   VAR
      s_FB_ItemError { ExternalAccessible := 'False'; ExternalVisible := 'False'; ExternalWritable := 'False'; S7_SetPoint := 'False'} : "FB_ItemError";   // Item error block's instance
      s_FB_ItemStatus { ExternalAccessible := 'False'; ExternalVisible := 'False'; ExternalWritable := 'False'; S7_SetPoint := 'False'} : "FB_ItemStatus";   // Item status block's instance
      ss_FIFOStatus { ExternalAccessible := 'False'; ExternalVisible := 'False'; ExternalWritable := 'False'; S7_SetPoint := 'False'} : "UDT_FifoStatus";   // Status structure
      s_UDT_Message { ExternalAccessible := 'False'; ExternalVisible := 'False'; ExternalWritable := 'False'; S7_SetPoint := 'False'} : "UDT_MessageV2";   // Message
      s_UDT_CodingBeltModesStatusOld { ExternalAccessible := 'False'; ExternalVisible := 'False'; ExternalWritable := 'False'; S7_SetPoint := 'False'} : "UDT_CodingBeltModesStatus";   // CodingBeltModes status structure
      s_UDT_ItemError { ExternalAccessible := 'False'; ExternalVisible := 'False'; ExternalWritable := 'False'; S7_SetPoint := 'False'} : "UDT_ItemError";   // Item error message body structure
      s_UDT_ItemStatus { ExternalAccessible := 'False'; ExternalVisible := 'False'; ExternalWritable := 'False'; S7_SetPoint := 'False'} : "UDT_ItemStatus";   // Item status message body structure
      s_R_TRIG_Connection {InstructionName := 'R_TRIG'; LibVersion := '1.0'; ExternalAccessible := 'False'; ExternalVisible := 'False'; ExternalWritable := 'False'; S7_SetPoint := 'False'} : R_TRIG;   // Rising edge trigger connection reastablished
      s_F_TRIG_SendAllErrors {InstructionName := 'F_TRIG'; LibVersion := '1.0'; ExternalAccessible := 'False'; ExternalVisible := 'False'; ExternalWritable := 'False'; S7_SetPoint := 'False'} : F_TRIG;   // Falling edge trigger from signal send all errors
      sdi_Code { ExternalAccessible := 'False'; ExternalVisible := 'False'; ExternalWritable := 'False'} : DInt;   // Error code
      si_ItemStatus { ExternalAccessible := 'False'; ExternalVisible := 'False'; ExternalWritable := 'False'} : Int;   // Item status
      ii_ErrorNumber { ExternalAccessible := 'False'; ExternalVisible := 'False'; ExternalWritable := 'False'} : Int;   // Counter Error Number
      si_State { ExternalAccessible := 'False'; ExternalVisible := 'False'; ExternalWritable := 'False'} : Int;   // Error state
      sx_ItemErrorMessageReq { ExternalAccessible := 'False'; ExternalVisible := 'False'; ExternalWritable := 'False'} : Bool;   // Item error message required
      sx_ItemStatusMessageReq { ExternalAccessible := 'False'; ExternalVisible := 'False'; ExternalWritable := 'False'} : Bool;   // Item status message required
      sx_SendAllProcedure { ExternalAccessible := 'False'; ExternalVisible := 'False'; ExternalWritable := 'False'} : Bool;   // Send all procedure
      sx_FIFOError { ExternalAccessible := 'False'; ExternalVisible := 'False'; ExternalWritable := 'False'} : Bool;   // FIFO error
      sx_FIFOWarning { ExternalAccessible := 'False'; ExternalVisible := 'False'; ExternalWritable := 'False'} : Bool;   // FIFO warning
      sx_ItemErrorBlockError { ExternalAccessible := 'False'; ExternalVisible := 'False'; ExternalWritable := 'False'} : Bool;   // Item error block error
      sx_ItemErrorBlockWarning { ExternalAccessible := 'False'; ExternalVisible := 'False'; ExternalWritable := 'False'} : Bool;   // Item error block warning
      sx_ItemStatusBlockError { ExternalAccessible := 'False'; ExternalVisible := 'False'; ExternalWritable := 'False'} : Bool;   // Item status block error
      sx_ItemStatusBlockWarning { ExternalAccessible := 'False'; ExternalVisible := 'False'; ExternalWritable := 'False'} : Bool;   // Item status block warning
   END_VAR


BEGIN
	(*
	----------------------------------------------------------------------------------------
	|                                                                                      |
	|  Copyright  2023             FORTNA Europe BV                                        |
	|  All Rights Reserved         Netherlands                                             |
	|                                                                                      |
	----------------------------------------------------------------------------------------
	Version history:
	Date        | Version   | Author       | Remark
	----------------------------------------------------------------------------------------
	26/04/2023  | 1.0       | M. Diebel   | Release TIA 17  | DHL Munich 2023
	06/10/2023  | 1.1       | M. Diebel   | Status handling | DHL Munich 2023
	13/03/2023  | 1.2       | S. Nieswiec  | Updated for new Baseline
	*)


	REGION 1 - Initialize message required signals

	    #sx_ItemErrorMessageReq := FALSE;
	    #sx_ItemStatusMessageReq := FALSE;

	    // On connection reestablish send last remembered status and error state ( status only when it's diffrent then 0 )
	    #s_R_TRIG_Connection(CLK := #ix_MFCConnected);

	    IF #s_R_TRIG_Connection.Q AND #si_ItemStatus <> 0
	    THEN
	        #sx_ItemStatusMessageReq := TRUE;
	    END_IF;

	    IF #s_R_TRIG_Connection.Q
	    THEN
	        #sx_ItemErrorMessageReq := TRUE;
	    END_IF;

	    // Prepare trigger on the collective reset signal.
	    #s_F_TRIG_SendAllErrors(CLK := #ix_SendAllErrorsState);

	    // When collective reset will go down, start send every equipment errors.
	    IF #s_F_TRIG_SendAllErrors.Q AND NOT #sx_SendAllProcedure
	    THEN
	        #ii_ErrorNumber := 0;
	        #sx_SendAllProcedure := TRUE;
	    END_IF;

	END_REGION

	REGION 2 - FIFO header status update

	    // Mode 'S' - FIFO register status update.
	    "FC_Fifo"(ic_Mode := 'S',
	              qUDT_Status => #ss_FIFOStatus,
	              qx_Error => #sx_FIFOError,
	              qx_Warning => #sx_FIFOWarning,
	              iqv_Data := #s_UDT_Message,
	              iqUDT_FifoHeader := #iq_UDT_FifoHeader,
	              iqv_DataBuffer := #iqs_FifoData);

	END_REGION

	REGION 3 - Prepare message data

	    // When there is no reset errors command, update errors.
	    IF NOT #ix_CollectiveReset
	        AND NOT #ss_FIFOStatus.FifoPreFull
	    THEN

	        // Status
	        IF (#i_UDT_CodingBeltModesStatus.Status <> #s_UDT_CodingBeltModesStatusOld.Status OR (#sx_SendAllProcedure AND #ii_ErrorNumber = 0))
	        THEN
	            #sx_ItemStatusMessageReq := TRUE;
	            #si_ItemStatus := #i_UDT_CodingBeltModesStatus.Status;
	            #s_UDT_CodingBeltModesStatusOld.Status := #i_UDT_CodingBeltModesStatus.Status;
	            #sx_SendAllProcedure := FALSE;
	        END_IF;


	        IF (#i_UDT_CodingBeltModesStatus.Specific.GeneralError <> #s_UDT_CodingBeltModesStatusOld.Specific.GeneralError AND NOT #sx_SendAllProcedure)
	            OR (#sx_SendAllProcedure AND #ii_ErrorNumber = 0)
	        THEN
	            #sdi_Code := "DB_MFC_ErrorCode".CodingBeltModes.GeneralError;
	            #si_State := BOOL_TO_INT(#i_UDT_CodingBeltModesStatus.Specific.GeneralError);
	            #s_UDT_CodingBeltModesStatusOld.Specific.GeneralError := #i_UDT_CodingBeltModesStatus.Specific.GeneralError;
	            #sx_ItemErrorMessageReq := TRUE;
	            #ii_ErrorNumber += 1;
	        ELSIF (#i_UDT_CodingBeltModesStatus.Specific.ConfigurationError <> #s_UDT_CodingBeltModesStatusOld.Specific.ConfigurationError AND NOT #sx_SendAllProcedure)
	            OR (#sx_SendAllProcedure AND #ii_ErrorNumber = 1)
	        THEN
	            #sdi_Code := "DB_MFC_ErrorCode".CodingBeltModes.ConfigurationError;
	            #si_State := BOOL_TO_INT(#i_UDT_CodingBeltModesStatus.Specific.ConfigurationError);
	            #s_UDT_CodingBeltModesStatusOld.Specific.ConfigurationError := #i_UDT_CodingBeltModesStatus.Specific.ConfigurationError;
	            #sx_ItemErrorMessageReq := TRUE;
	            #ii_ErrorNumber += 1;
	            #sx_SendAllProcedure := FALSE;
	        END_IF;

	    END_IF;

	END_REGION

	REGION 4 - Write message components to the item error structure

	    #s_UDT_ItemError.ItemNumber := #i_UDT_EquipmentNumber;
	    #s_UDT_ItemError.Error := #sdi_Code;
	    #s_UDT_ItemError.State := #si_State;
	    #s_UDT_ItemError.Masked := 1;

	END_REGION

	REGION 5 - Write message components to the item status structure

	    #s_UDT_ItemStatus.Group := #i_UDT_EquipmentNumber.Group;
	    #s_UDT_ItemStatus.Node := #i_UDT_EquipmentNumber.Node;
	    #s_UDT_ItemStatus.Status := #si_ItemStatus;

	END_REGION

	REGION 6 - Prepare messages to the MFC

	    // If item error message required signal is set, prepare the item error message.
	    IF (#sx_ItemErrorMessageReq)
	    THEN
	        #s_FB_ItemError(i_UDT_ItemErrorBody := #s_UDT_ItemError,
	                        ii_MessageGroup := 1,
	                        ix_FlagRetry := FALSE,
	                        idi_TimeSpan := 0,
	                        qx_Error => #sx_ItemErrorBlockError,
	                        qx_Warning => #sx_ItemErrorBlockWarning,
	                        iq_UDT_FifoHeader := #iq_UDT_FifoHeader,
	                        iqs_FifoData := #iqs_FifoData,
	                        iqdi_MessageSequenceNumber := #iqdi_MessageSequenceNumber);
	    END_IF;

	    // If item status message required signal is set, prepare the item error message.
	    IF (#sx_ItemStatusMessageReq)
	    THEN
	        #s_FB_ItemStatus(i_UDT_ItemStatusBody := #s_UDT_ItemStatus,
	                         ii_MessageGroup := 1,
	                         ix_FlagRetry := FALSE,
	                         idi_TimeSpan := 0,
	                         qx_Error => #sx_ItemStatusBlockError,
	                         qx_Warning => #sx_ItemStatusBlockWarning,
	                         iq_UDT_FifoHeader := #iq_UDT_FifoHeader,
	                         iqs_FifoData := #iqs_FifoData,
	                         iqdi_MessageSequenceNumber := #iqdi_MessageSequenceNumber);
	    END_IF;

	END_REGION

	REGION 7 - Write outputs

	    // Prepare collective output error.
	    #qx_Error :=
	    #sx_ItemErrorBlockError
	    OR #sx_ItemStatusBlockError
	    OR #sx_FIFOError;

	    // Prepare collective output warning.
	    #qx_Warning :=
	    #sx_ItemErrorBlockWarning
	    OR #sx_ItemStatusBlockWarning
	    OR #sx_FIFOWarning;

	END_REGION




END_FUNCTION_BLOCK

FUNCTION_BLOCK "FB_MFC_Visu_PECUpdate_Status"
{ S7_Optimized_Access := 'TRUE' }
VERSION : 2.0
// ATTRIBUTES
// AUTO_NUMBER = True
// BLOCK_NUMBER = 249
// END_ATTRIBUTES
   VAR_INPUT
      ix_SendAllErrorsState { ExternalAccessible := 'False'; ExternalVisible := 'False'; ExternalWritable := 'False'} : Bool;   // True - update all the messages
      ix_MFCConnected { ExternalAccessible := 'False'; ExternalVisible := 'False'; ExternalWritable := 'False'} : Bool;   // True - A connection to the MFC has been established
      ix_CollectiveReset { ExternalAccessible := 'False'; ExternalVisible := 'False'; ExternalWritable := 'False'} : Bool;   // True - Collective reset command of all system controls
      i_UDT_PECUpdateStatus { ExternalAccessible := 'False'; ExternalVisible := 'False'; ExternalWritable := 'False'} : "UDT_PECUpdateStatus";   // Input PEC update status structrue
      i_UDT_EquipmentNumber { ExternalAccessible := 'False'; ExternalVisible := 'False'; ExternalWritable := 'False'} : "UDT_EquipmentNumber";   // Item number
   END_VAR

   VAR_OUTPUT
      qx_Error { ExternalAccessible := 'False'; ExternalVisible := 'False'; ExternalWritable := 'False'} : Bool;   // Block error
      qx_Warning { ExternalAccessible := 'False'; ExternalVisible := 'False'; ExternalWritable := 'False'} : Bool;   // Block warning
   END_VAR

   VAR_IN_OUT
      iq_UDT_FifoHeader : "UDT_FifoHeader";   // FIFO header
      iqs_FifoData : Array[*] of "UDT_MessageV2";   // FIFO data buffer
      iqdi_MessageSequenceNumber { ExternalAccessible := 'False'; ExternalVisible := 'False'; ExternalWritable := 'False'} : DInt;   // Message number
   END_VAR

   VAR
      s_FB_ItemError { ExternalAccessible := 'False'; ExternalVisible := 'False'; ExternalWritable := 'False'; S7_SetPoint := 'False'} : "FB_ItemError";   // Item error block's instance
      s_FB_TIDLost { ExternalAccessible := 'False'; ExternalVisible := 'False'; ExternalWritable := 'False'; S7_SetPoint := 'False'} : "FB_TIDLost";   // TID lost message block instance
      s_UDT_PECUpdateOLD { ExternalAccessible := 'False'; ExternalVisible := 'False'; ExternalWritable := 'False'; S7_SetPoint := 'False'} : "UDT_PECUpdateStatus";   // PEC Update old status structure
      s_UDT_PECUpdate { ExternalAccessible := 'False'; ExternalVisible := 'False'; ExternalWritable := 'False'; S7_SetPoint := 'False'} : "UDT_PECUpdateStatus";   // PEC Update status structure
      s_UDT_ItemError { ExternalAccessible := 'False'; ExternalVisible := 'False'; ExternalWritable := 'False'; S7_SetPoint := 'False'} : "UDT_ItemError";   // Item error message body structure
      s_UDT_FIFOStatus { ExternalAccessible := 'False'; ExternalVisible := 'False'; ExternalWritable := 'False'; S7_SetPoint := 'False'} : "UDT_FifoStatus";   // FIFO status structure
      s_UDT_Message { ExternalAccessible := 'False'; ExternalVisible := 'False'; ExternalWritable := 'False'; S7_SetPoint := 'False'} : "UDT_BytesMessage";   // Message
      s_R_TRIG_Connection {InstructionName := 'R_TRIG'; LibVersion := '1.0'; ExternalAccessible := 'False'; ExternalVisible := 'False'; ExternalWritable := 'False'; S7_SetPoint := 'False'} : R_TRIG;   // Connection reestablished
      s_F_TRIG_SendAllErrors {InstructionName := 'F_TRIG'; LibVersion := '1.0'; ExternalAccessible := 'False'; ExternalVisible := 'False'; ExternalWritable := 'False'; S7_SetPoint := 'False'} : F_TRIG;
      ss_TIDLostReason { ExternalAccessible := 'False'; ExternalVisible := 'False'; ExternalWritable := 'False'} : Struct   // TID lost message reason
         Unknown { ExternalAccessible := 'False'; ExternalVisible := 'False'; ExternalWritable := 'False'} : Bool;   //        Unknown
         TIDLost { ExternalAccessible := 'False'; ExternalVisible := 'False'; ExternalWritable := 'False'} : Bool;   //        TID lost
         EndOfLine { ExternalAccessible := 'False'; ExternalVisible := 'False'; ExternalWritable := 'False'} : Bool;   //        End of line
         ParcelDidntArrive { ExternalAccessible := 'False'; ExternalVisible := 'False'; ExternalWritable := 'False'} : Bool;   //        Parcel didn't arrave on PEC when expected
         UserDelete { ExternalAccessible := 'False'; ExternalVisible := 'False'; ExternalWritable := 'False'} : Bool;   //        User delete
      END_STRUCT;
      sdi_Code { ExternalAccessible := 'False'; ExternalVisible := 'False'; ExternalWritable := 'False'} : DInt;   // Error code
      si_ItemStatus { ExternalAccessible := 'False'; ExternalVisible := 'False'; ExternalWritable := 'False'} : Int;   // Item status
      si_State { ExternalAccessible := 'False'; ExternalVisible := 'False'; ExternalWritable := 'False'} : Int;   // Error state
      ii_ErrorNumber { ExternalAccessible := 'False'; ExternalVisible := 'False'; ExternalWritable := 'False'} : Int;
      sx_ItemErrorMessageReq { ExternalAccessible := 'False'; ExternalVisible := 'False'; ExternalWritable := 'False'} : Bool;   // Item error message required
      sx_ItemErrorBlockError { ExternalAccessible := 'False'; ExternalVisible := 'False'; ExternalWritable := 'False'} : Bool;   // Item error block error
      sx_FIFOError { ExternalAccessible := 'False'; ExternalVisible := 'False'; ExternalWritable := 'False'} : Bool;   // FIFO error
      sx_FIFOWarning { ExternalAccessible := 'False'; ExternalVisible := 'False'; ExternalWritable := 'False'} : Bool;   // FIFO warning
      sx_ItemErrorBlockWarning { ExternalAccessible := 'False'; ExternalVisible := 'False'; ExternalWritable := 'False'} : Bool;   // Item error block warning
      sx_SendAllProcedure { ExternalAccessible := 'False'; ExternalVisible := 'False'; ExternalWritable := 'False'} : Bool;
   END_VAR

   VAR_TEMP
      ti_GINLost : Int;   //        Lost GIN
      ti_LC_TIDLost : Int;   //        FIFO check for GIN lost
   END_VAR


BEGIN
	(*
	----------------------------------------------------------------------------------------
	|                                                                                      |
	|  Copyright  2023             FORTNA Europe BV                                        |
	|  All Rights Reserved         Netherlands                                             |
	|                                                                                      |
	----------------------------------------------------------------------------------------
	Version history:
	Date        | Version   | Author       | Remark
	----------------------------------------------------------------------------------------
	03/01/2023  | 1.0       | S. Nikodem   | Release TIA 17 | DHL Munich 2023
	10/08/2023  | 2.0       | M. Diebel    | Copy input data to static memory | DHL Munich 2023
	13/03/2023  | 2.1       | S. Nieswiec  | Updated for new Baseline
	*)

	// To check line 76 - relation to DB_GIN, in Malmo they updated UDT_GIN

	REGION 1 - Initialize message required signals

	    #sx_ItemErrorMessageReq := FALSE;

	    // On connection reestablish send last remembered status and error state ( status only when it's diffrent then 0 )
	    #s_R_TRIG_Connection(CLK := #ix_MFCConnected);

	    // Prepare trigger on the collective reset signal.
	    #s_F_TRIG_SendAllErrors(CLK := #ix_SendAllErrorsState);

	    // When collective reset will go down, start send every equipment errors.
	    IF #s_F_TRIG_SendAllErrors.Q AND NOT #sx_SendAllProcedure
	    THEN
	        #ii_ErrorNumber := 0;
	        #sx_SendAllProcedure := TRUE;
	    END_IF;

	END_REGION

	REGION 2 - FIFO header status update

	    // Mode 'S' - FIFO register status update.
	    "FC_Fifo"(ic_Mode := 'S',
	              qUDT_Status => #s_UDT_FIFOStatus,
	              qx_Error => #sx_FIFOError,
	              qx_Warning => #sx_FIFOWarning,
	              iqv_Data := #s_UDT_Message,
	              iqUDT_FifoHeader := #iq_UDT_FifoHeader,
	              iqv_DataBuffer := #iqs_FifoData);

	END_REGION

	REGION 3 - Prepare message data

	    // When there is no reset errors command, update status and errors.
	    IF NOT #ix_CollectiveReset
	        AND NOT #s_UDT_FIFOStatus.FifoPreFull
	    THEN

	        //Copy input data to static memory
	        #s_UDT_PECUpdate := #i_UDT_PECUpdateStatus;

	        // If the status changed, set item error message required signal.
	        IF (#s_UDT_PECUpdate <> #s_UDT_PECUpdateOLD OR #sx_SendAllProcedure)
	        THEN
	            #sx_ItemErrorMessageReq := TRUE;

	            // Check which specific status changed, prepare code, change state and write new status into the old one.
	            IF (#s_UDT_PECUpdate.LowPerformance <> #s_UDT_PECUpdateOLD.LowPerformance AND NOT #sx_SendAllProcedure)
	                OR (#sx_SendAllProcedure AND #ii_ErrorNumber = 0)
	            THEN
	                #sdi_Code := "DB_MFC_ErrorCode".PECUpdate.LowPerformance;
	                #si_State := BOOL_TO_INT(#s_UDT_PECUpdate.LowPerformance);
	                #s_UDT_PECUpdateOLD.LowPerformance := #s_UDT_PECUpdate.LowPerformance;
	                #ii_ErrorNumber += 1;
	            ELSIF (#s_UDT_PECUpdate.TooManyLost <> #s_UDT_PECUpdateOLD.TooManyLost AND NOT #sx_SendAllProcedure)
	                OR (#sx_SendAllProcedure AND #ii_ErrorNumber = 1)
	            THEN
	                #sdi_Code := "DB_MFC_ErrorCode".PECUpdate.TooManyLost;
	                #si_State := BOOL_TO_INT(#s_UDT_PECUpdate.TooManyLost);
	                #s_UDT_PECUpdateOLD.TooManyLost := #s_UDT_PECUpdate.TooManyLost;
	                #ii_ErrorNumber += 1;
	            ELSIF (#s_UDT_PECUpdate.PEC <> #s_UDT_PECUpdateOLD.PEC)
	            THEN
	                #sx_ItemErrorMessageReq := FALSE;
	                #s_UDT_PECUpdateOLD.PEC := #s_UDT_PECUpdate.PEC;
	            ELSIF (#s_UDT_PECUpdate.Jam <> #s_UDT_PECUpdateOLD.Jam AND NOT #sx_SendAllProcedure)
	                OR (#sx_SendAllProcedure AND #ii_ErrorNumber = 2)
	            THEN
	                #sdi_Code := "DB_MFC_ErrorCode".PECUpdate.Jam;
	                #si_State := BOOL_TO_INT(#s_UDT_PECUpdate.Jam);
	                #s_UDT_PECUpdateOLD.Jam := #s_UDT_PECUpdate.Jam;
	                #sx_SendAllProcedure := FALSE;
	            END_IF;

	        END_IF;

	    END_IF;

	END_REGION

	REGION 4 - Write message components to the item error structure

	    #s_UDT_ItemError.ItemNumber := #i_UDT_EquipmentNumber;
	    #s_UDT_ItemError.Error := #sdi_Code;
	    #s_UDT_ItemError.State := #si_State;
	    #s_UDT_ItemError.Masked := 1;

	END_REGION

	REGION 5 - Prepare messages to the MFC

	    // If item error message required signal is set, prepare the item error message.
	    IF (#sx_ItemErrorMessageReq)
	    THEN
	        #s_FB_ItemError(i_UDT_ItemErrorBody := #s_UDT_ItemError,
	                        ii_MessageGroup := 1,
	                        ix_FlagRetry := FALSE,
	                        qx_Error => #sx_ItemErrorBlockError,
	                        qx_Warning => #sx_ItemErrorBlockWarning,
	                        iq_UDT_FifoHeader := #iq_UDT_FifoHeader,
	                        iqs_FifoData := #iqs_FifoData,
	                        iqdi_MessageSequenceNumber := #iqdi_MessageSequenceNumber);
	    END_IF;

	END_REGION

	REGION 6 - Write outputs

	    // Prepare collective output error.
	    #qx_Error := #sx_ItemErrorBlockError
	    OR #sx_FIFOError;

	    // Prepare collective output warning.
	    #qx_Warning := #sx_ItemErrorBlockWarning
	    OR #sx_FIFOWarning;

	END_REGION
END_FUNCTION_BLOCK

FUNCTION_BLOCK "FB_MFC_Visu_Connect_Status"
{ S7_Optimized_Access := 'TRUE' }
VERSION : 0.1
// ATTRIBUTES
// AUTO_NUMBER = True
// BLOCK_NUMBER = 140
// END_ATTRIBUTES
   VAR_INPUT
      i_UDT_ConnectStatus { ExternalAccessible := 'False'; ExternalVisible := 'False'; ExternalWritable := 'False'} : "UDT_ConnectStatus";   // TCPIPConnection status structure
      i_UDT_EquipmentNumber { ExternalAccessible := 'False'; ExternalVisible := 'False'; ExternalWritable := 'False'} : "UDT_EquipmentNumber";   // Item number
      ix_SendAllErrorsState { ExternalAccessible := 'False'; ExternalVisible := 'False'; ExternalWritable := 'False'} : Bool;   // True - update all the messages
      ix_MFCConnected { ExternalAccessible := 'False'; ExternalVisible := 'False'; ExternalWritable := 'False'} : Bool;   // True - A connection to the MFC has been established
      ix_CollectiveReset { ExternalAccessible := 'False'; ExternalVisible := 'False'; ExternalWritable := 'False'} : Bool;   // True - Collective reset command of all system controls
   END_VAR

   VAR_OUTPUT
      qx_Error { ExternalAccessible := 'False'; ExternalVisible := 'False'; ExternalWritable := 'False'} : Bool;   // Block error
      qx_Warning { ExternalAccessible := 'False'; ExternalVisible := 'False'; ExternalWritable := 'False'} : Bool;   // Block warning
   END_VAR

   VAR_IN_OUT
      iq_UDT_FifoHeader : "UDT_FifoHeader";   // FIFO header
      iqs_FifoData : Array[*] of "UDT_MessageV2";   // FIFO data buffer
      iqdi_MessageSequenceNumber { ExternalAccessible := 'False'; ExternalVisible := 'False'; ExternalWritable := 'False'} : DInt;   // Message number
   END_VAR

   VAR
      s_FB_ItemError { ExternalAccessible := 'False'; ExternalVisible := 'False'; ExternalWritable := 'False'; S7_SetPoint := 'False'} : "FB_ItemError";   // Item error block's instance
      s_FB_ItemStatus { ExternalAccessible := 'False'; ExternalVisible := 'False'; ExternalWritable := 'False'; S7_SetPoint := 'False'} : "FB_ItemStatus";   // Item status block's instance
      ss_FIFOStatus { ExternalAccessible := 'False'; ExternalVisible := 'False'; ExternalWritable := 'False'; S7_SetPoint := 'False'} : "UDT_FifoStatus";   // Status structure
      s_UDT_Message { ExternalAccessible := 'False'; ExternalVisible := 'False'; ExternalWritable := 'False'; S7_SetPoint := 'False'} : "UDT_MessageV2";   // Message
      s_UDT_ConnectStatusOld { ExternalAccessible := 'False'; ExternalVisible := 'False'; ExternalWritable := 'False'; S7_SetPoint := 'False'} : "UDT_ConnectStatus";   // TCPIPConnection status structure
      s_UDT_ItemError { ExternalAccessible := 'False'; ExternalVisible := 'False'; ExternalWritable := 'False'; S7_SetPoint := 'False'} : "UDT_ItemError";   // Item error message body structure
      s_UDT_ItemStatus { ExternalAccessible := 'False'; ExternalVisible := 'False'; ExternalWritable := 'False'; S7_SetPoint := 'False'} : "UDT_ItemStatus";   // Item status message body structure
      s_R_TRIG_Connection {InstructionName := 'R_TRIG'; LibVersion := '1.0'; ExternalAccessible := 'False'; ExternalVisible := 'False'; ExternalWritable := 'False'; S7_SetPoint := 'False'} : R_TRIG;   // Rising edge trigger connection reastablished
      s_F_TRIG_SendAllErrors {InstructionName := 'F_TRIG'; LibVersion := '1.0'; ExternalAccessible := 'False'; ExternalVisible := 'False'; ExternalWritable := 'False'; S7_SetPoint := 'False'} : F_TRIG;   // Falling edge trigger from signal send all errors
      sdi_Code { ExternalAccessible := 'False'; ExternalVisible := 'False'; ExternalWritable := 'False'} : DInt;   // Error code
      si_ItemStatus { ExternalAccessible := 'False'; ExternalVisible := 'False'; ExternalWritable := 'False'} : Int;   // Item status
      ii_ErrorNumber { ExternalAccessible := 'False'; ExternalVisible := 'False'; ExternalWritable := 'False'} : Int;   // Counter Error Number
      si_State { ExternalAccessible := 'False'; ExternalVisible := 'False'; ExternalWritable := 'False'} : Int;   // Error state
      sx_ItemErrorMessageReq { ExternalAccessible := 'False'; ExternalVisible := 'False'; ExternalWritable := 'False'} : Bool;   // Item error message required
      sx_ItemStatusMessageReq { ExternalAccessible := 'False'; ExternalVisible := 'False'; ExternalWritable := 'False'} : Bool;   // Item status message required
      sx_SendAllProcedure { ExternalAccessible := 'False'; ExternalVisible := 'False'; ExternalWritable := 'False'} : Bool;   // Send all procedure
      sx_FIFOError { ExternalAccessible := 'False'; ExternalVisible := 'False'; ExternalWritable := 'False'} : Bool;   // FIFO error
      sx_FIFOWarning { ExternalAccessible := 'False'; ExternalVisible := 'False'; ExternalWritable := 'False'} : Bool;   // FIFO warning
      sx_ItemErrorBlockError { ExternalAccessible := 'False'; ExternalVisible := 'False'; ExternalWritable := 'False'} : Bool;   // Item error block error
      sx_ItemErrorBlockWarning { ExternalAccessible := 'False'; ExternalVisible := 'False'; ExternalWritable := 'False'} : Bool;   // Item error block warning
      sx_ItemStatusBlockError { ExternalAccessible := 'False'; ExternalVisible := 'False'; ExternalWritable := 'False'} : Bool;   // Item status block error
      sx_ItemStatusBlockWarning { ExternalAccessible := 'False'; ExternalVisible := 'False'; ExternalWritable := 'False'} : Bool;   // Item status block warning
   END_VAR


BEGIN
	(*
	----------------------------------------------------------------------------------------
	|                                                                                      |
	|  Copyright  2023             FORTNA Europe BV                                        |
	|  All Rights Reserved         Netherlands                                             |
	|                                                                                      |
	----------------------------------------------------------------------------------------
	Version history:
	Date        | Version   | Author       | Remark
	----------------------------------------------------------------------------------------
	31/03/2023  | 1.0       | M. Diebel   | Release TIA 17 | DHL Munich 2023
	13/03/2023  | 1.1       | S. Nieswiec | Updated for new Baseline
	*)


	REGION 1 - Initialize message required signals

	    #sx_ItemErrorMessageReq := FALSE;
	    #sx_ItemStatusMessageReq := FALSE;

	    // On connection reestablish send last remembered status and error state ( status only when it's diffrent then 0 )
	    #s_R_TRIG_Connection(CLK := #ix_MFCConnected);

	    IF #s_R_TRIG_Connection.Q AND #si_ItemStatus <> 0
	    THEN
	        #sx_ItemStatusMessageReq := TRUE;
	    END_IF;

	    IF #s_R_TRIG_Connection.Q
	    THEN
	        #sx_ItemErrorMessageReq := TRUE;
	    END_IF;

	    // Prepare trigger on the collective reset signal.
	    #s_F_TRIG_SendAllErrors(CLK := #ix_SendAllErrorsState);

	    // When collective reset will go down, start send every equipment errors.
	    IF #s_F_TRIG_SendAllErrors.Q AND NOT #sx_SendAllProcedure
	    THEN
	        #ii_ErrorNumber := 0;
	        #sx_SendAllProcedure := TRUE;
	    END_IF;

	END_REGION

	REGION 2 - FIFO header status update

	    // Mode 'S' - FIFO register status update.
	    "FC_Fifo"(ic_Mode := 'S',
	              qUDT_Status => #ss_FIFOStatus,
	              qx_Error => #sx_FIFOError,
	              qx_Warning => #sx_FIFOWarning,
	              iqv_Data := #s_UDT_Message,
	              iqUDT_FifoHeader := #iq_UDT_FifoHeader,
	              iqv_DataBuffer := #iqs_FifoData);

	END_REGION

	REGION 3 - Prepare message data

	    // When there is no reset errors command, update status and errors.
	    IF NOT #ix_CollectiveReset
	        AND NOT #ss_FIFOStatus.FifoPreFull
	    THEN
	        // Status
	        IF (#i_UDT_ConnectStatus.Status <> #s_UDT_ConnectStatusOld.Status OR (#sx_SendAllProcedure AND #ii_ErrorNumber = 0))
	        THEN
	            #sx_ItemStatusMessageReq := TRUE;
	            #si_ItemStatus := #i_UDT_ConnectStatus.Status;
	            #s_UDT_ConnectStatusOld.Status := #i_UDT_ConnectStatus.Status;
	        END_IF;


	        // Check which specific status changed, prepare code, change state and write new status into the old one.
	        IF (#i_UDT_ConnectStatus.Specific.CommunicationFault <> #s_UDT_ConnectStatusOld.Specific.CommunicationFault AND NOT #sx_SendAllProcedure)
	            OR (#sx_SendAllProcedure AND #ii_ErrorNumber = 0)
	        THEN
	            #sdi_Code := "DB_MFC_ErrorCode".Connect.CommunicationFault;
	            #si_State := BOOL_TO_INT(#i_UDT_ConnectStatus.Specific.CommunicationFault);
	            #s_UDT_ConnectStatusOld.Specific.CommunicationFault := #i_UDT_ConnectStatus.Specific.CommunicationFault;
	            #sx_ItemErrorMessageReq := TRUE;
	            #sx_SendAllProcedure := FALSE;
	        END_IF;
	    END_IF;
	END_REGION

	REGION 4 - Write message components to the item error structure

	    #s_UDT_ItemError.ItemNumber := #i_UDT_EquipmentNumber;
	    #s_UDT_ItemError.Error := #sdi_Code;
	    #s_UDT_ItemError.State := #si_State;
	    #s_UDT_ItemError.Masked := 1;

	END_REGION

	REGION 5 - Write message components to the item status structure

	    #s_UDT_ItemStatus.Group := #i_UDT_EquipmentNumber.Group;
	    #s_UDT_ItemStatus.Node := #i_UDT_EquipmentNumber.Node;
	    #s_UDT_ItemStatus.Status := #si_ItemStatus;

	END_REGION

	REGION 6 - Prepare messages to the MFC

	    // If item error message required signal is set, prepare the item error message.
	    IF (#sx_ItemErrorMessageReq)
	    THEN
	        #s_FB_ItemError(i_UDT_ItemErrorBody := #s_UDT_ItemError,
	                        ii_MessageGroup := 1,
	                        ix_FlagRetry := FALSE,
	                        idi_TimeSpan := 0,
	                        qx_Error => #sx_ItemErrorBlockError,
	                        qx_Warning => #sx_ItemErrorBlockWarning,
	                        iq_UDT_FifoHeader := #iq_UDT_FifoHeader,
	                        iqs_FifoData := #iqs_FifoData,
	                        iqdi_MessageSequenceNumber := #iqdi_MessageSequenceNumber);
	    END_IF;

	    // If item status message required signal is set, prepare the item error message.
	    IF (#sx_ItemStatusMessageReq)
	    THEN
	        #s_FB_ItemStatus(i_UDT_ItemStatusBody := #s_UDT_ItemStatus,
	                         ii_MessageGroup := 1,
	                         ix_FlagRetry := FALSE,
	                         idi_TimeSpan := 0,
	                         qx_Error => #sx_ItemStatusBlockError,
	                         qx_Warning => #sx_ItemStatusBlockWarning,
	                         iq_UDT_FifoHeader := #iq_UDT_FifoHeader,
	                         iqs_FifoData := #iqs_FifoData,
	                         iqdi_MessageSequenceNumber := #iqdi_MessageSequenceNumber);
	    END_IF;

	END_REGION

	REGION 7 - Write outputs

	    // Prepare collective output error.
	    #qx_Error :=
	    #sx_ItemErrorBlockError
	    OR #sx_ItemStatusBlockError
	    OR #sx_FIFOError;

	    // Prepare collective output warning.
	    #qx_Warning :=
	    #sx_ItemErrorBlockWarning
	    OR #sx_ItemStatusBlockWarning
	    OR #sx_FIFOWarning;

	END_REGION



END_FUNCTION_BLOCK

FUNCTION_BLOCK "FB_MFC_Visu_Outfeed2States_Status"
{ S7_Optimized_Access := 'TRUE' }
VERSION : 2.0
// ATTRIBUTES
// AUTO_NUMBER = True
// BLOCK_NUMBER = 152
// END_ATTRIBUTES
   VAR_INPUT
      i_UDT_Outfeed2StatesStatus { ExternalAccessible := 'False'; ExternalVisible := 'False'; ExternalWritable := 'False'} : "UDT_Outfeed2StatesStatus";   // Outfeed2States status structure
      i_UDT_EquipmentNumber { ExternalAccessible := 'False'; ExternalVisible := 'False'; ExternalWritable := 'False'} : "UDT_EquipmentNumber";   // Item number
      ix_SendAllErrorsState { ExternalAccessible := 'False'; ExternalVisible := 'False'; ExternalWritable := 'False'} : Bool;   // True - update all the messages
      ix_MFCConnected { ExternalAccessible := 'False'; ExternalVisible := 'False'; ExternalWritable := 'False'} : Bool;   // True - A connection to the MFC has been established
      ix_CollectiveReset { ExternalAccessible := 'False'; ExternalVisible := 'False'; ExternalWritable := 'False'} : Bool;   // True - Collective reset command of all system controls
   END_VAR

   VAR_OUTPUT
      qx_Error { ExternalAccessible := 'False'; ExternalVisible := 'False'; ExternalWritable := 'False'} : Bool;   // Block error
      qx_Warning { ExternalAccessible := 'False'; ExternalVisible := 'False'; ExternalWritable := 'False'} : Bool;   // Block warning
   END_VAR

   VAR_IN_OUT
      iq_UDT_FifoHeader : "UDT_FifoHeader";   // FIFO header
      iqs_FifoData : Array[*] of "UDT_MessageV2";   // FIFO data buffer
      iqdi_MessageSequenceNumber { ExternalAccessible := 'False'; ExternalVisible := 'False'; ExternalWritable := 'False'} : DInt;   // Message number
   END_VAR

   VAR
      s_FB_ItemError { ExternalAccessible := 'False'; ExternalVisible := 'False'; ExternalWritable := 'False'; S7_SetPoint := 'False'} : "FB_ItemError";   // Item error block's instance
      s_FB_ItemStatus { ExternalAccessible := 'False'; ExternalVisible := 'False'; ExternalWritable := 'False'; S7_SetPoint := 'False'} : "FB_ItemStatus";   // Item status block's instance
      ss_FIFOStatus { ExternalAccessible := 'False'; ExternalVisible := 'False'; ExternalWritable := 'False'; S7_SetPoint := 'False'} : "UDT_FifoStatus";   // Status structure
      s_UDT_Message { ExternalAccessible := 'False'; ExternalVisible := 'False'; ExternalWritable := 'False'; S7_SetPoint := 'False'} : "UDT_MessageV2";   // Message
      s_UDT_Outfeed2StatesStatusOld { ExternalAccessible := 'False'; ExternalVisible := 'False'; ExternalWritable := 'False'; S7_SetPoint := 'False'} : "UDT_Outfeed2StatesStatus";   // Outfeed2States old status structure
      s_UDT_ItemError { ExternalAccessible := 'False'; ExternalVisible := 'False'; ExternalWritable := 'False'; S7_SetPoint := 'False'} : "UDT_ItemError";   // Item error message body structure
      s_UDT_ItemStatus { ExternalAccessible := 'False'; ExternalVisible := 'False'; ExternalWritable := 'False'; S7_SetPoint := 'False'} : "UDT_ItemStatus";   // Item status message body structure
      s_R_TRIG_Connection {InstructionName := 'R_TRIG'; LibVersion := '1.0'; ExternalAccessible := 'False'; ExternalVisible := 'False'; ExternalWritable := 'False'; S7_SetPoint := 'False'} : R_TRIG;   // Rising edge trigger connection reastablished
      s_F_TRIG_SendAllErrors {InstructionName := 'F_TRIG'; LibVersion := '1.0'; ExternalAccessible := 'False'; ExternalVisible := 'False'; ExternalWritable := 'False'; S7_SetPoint := 'False'} : F_TRIG;   // Falling edge trigger from signal send all errors
      sdi_Code { ExternalAccessible := 'False'; ExternalVisible := 'False'; ExternalWritable := 'False'} : DInt;   // Error code
      si_ItemStatus { ExternalAccessible := 'False'; ExternalVisible := 'False'; ExternalWritable := 'False'} : Int;   // Item status
      ii_ErrorNumber { ExternalAccessible := 'False'; ExternalVisible := 'False'; ExternalWritable := 'False'} : Int;   // Counter Error Number
      si_State { ExternalAccessible := 'False'; ExternalVisible := 'False'; ExternalWritable := 'False'} : Int;   // Error state
      sx_ItemErrorMessageReq { ExternalAccessible := 'False'; ExternalVisible := 'False'; ExternalWritable := 'False'} : Bool;   // Item error message required
      sx_ItemStatusMessageReq { ExternalAccessible := 'False'; ExternalVisible := 'False'; ExternalWritable := 'False'} : Bool;   // Item status message required
      sx_SendAllProcedure { ExternalAccessible := 'False'; ExternalVisible := 'False'; ExternalWritable := 'False'} : Bool;   // Send all procedure
      sx_FIFOError { ExternalAccessible := 'False'; ExternalVisible := 'False'; ExternalWritable := 'False'} : Bool;   // FIFO error
      sx_FIFOWarning { ExternalAccessible := 'False'; ExternalVisible := 'False'; ExternalWritable := 'False'} : Bool;   // FIFO warning
      sx_ItemErrorBlockError { ExternalAccessible := 'False'; ExternalVisible := 'False'; ExternalWritable := 'False'} : Bool;   // Item error block error
      sx_ItemErrorBlockWarning { ExternalAccessible := 'False'; ExternalVisible := 'False'; ExternalWritable := 'False'} : Bool;   // Item error block warning
      sx_ItemStatusBlockError { ExternalAccessible := 'False'; ExternalVisible := 'False'; ExternalWritable := 'False'} : Bool;   // Item status block error
      sx_ItemStatusBlockWarning { ExternalAccessible := 'False'; ExternalVisible := 'False'; ExternalWritable := 'False'} : Bool;   // Item status block warning
   END_VAR

   VAR_TEMP
      t_UDT_Outfeed2StatesStatus : "UDT_Outfeed2StatesStatus";   // Outfeed2States status structure
   END_VAR


BEGIN
	(*
	----------------------------------------------------------------------------------------
	|                                                                                      |
	|  Copyright  2023             FORTNA Europe BV                                        |
	|  All Rights Reserved         Netherlands                                             |
	|                                                                                      |
	----------------------------------------------------------------------------------------
	Version history:
	Date        | Version   | Author       | Remark
	----------------------------------------------------------------------------------------
	27/03/2023  | 1.0       | M. Diebel   | Release TIA 17 | DHL Munich 2023
	11/09/2023  | 2.0       | M. Diebel   | Disable the information messages to MFC
	13/03/2023  | 2.1       | S. Nieswiec | Updated for new Baseline
	*)


	REGION 1 - Initialize message required signals

	    #sx_ItemErrorMessageReq := FALSE;
	    #sx_ItemStatusMessageReq := FALSE;

	    //Move input to temp
	    #t_UDT_Outfeed2StatesStatus := #i_UDT_Outfeed2StatesStatus;
	    //Disable the information messages
	    //-ChuteFull
	    //-ChuteHalfFull
	    #t_UDT_Outfeed2StatesStatus.Specific.ChuteFull := FALSE;
	    #t_UDT_Outfeed2StatesStatus.Specific.ChuteHalfFull := FALSE;


	    // Prepare trigger on the collective reset signal.
	    #s_F_TRIG_SendAllErrors(CLK := #ix_SendAllErrorsState);

	    // When collective reset will go down, start send every equipment errors.
	    IF #s_F_TRIG_SendAllErrors.Q AND NOT #sx_SendAllProcedure
	    THEN
	        #ii_ErrorNumber := 0;
	        #sx_SendAllProcedure := TRUE;
	    END_IF;

	END_REGION

	REGION 2 - FIFO header status update

	    // Mode 'S' - FIFO register status update.
	    "FC_Fifo"(ic_Mode := 'S',
	              qUDT_Status => #ss_FIFOStatus,
	              qx_Error => #sx_FIFOError,
	              qx_Warning => #sx_FIFOWarning,
	              iqv_Data := #s_UDT_Message,
	              iqUDT_FifoHeader := #iq_UDT_FifoHeader,
	              iqv_DataBuffer := #iqs_FifoData);

	END_REGION

	REGION 3 - Prepare message data

	    // When there is no reset errors command, update status and errors.
	    IF NOT #ix_CollectiveReset
	        AND NOT #ss_FIFOStatus.FifoPreFull
	    THEN
	        // Status
	        IF (#t_UDT_Outfeed2StatesStatus.Status <> #s_UDT_Outfeed2StatesStatusOld.Status OR (#sx_SendAllProcedure AND #ii_ErrorNumber = 0))
	        THEN
	            #sx_ItemStatusMessageReq := TRUE;
	            #si_ItemStatus := #t_UDT_Outfeed2StatesStatus.Status;
	            #s_UDT_Outfeed2StatesStatusOld.Status := #t_UDT_Outfeed2StatesStatus.Status;
	        END_IF;

	        // Check which specific status changed, prepare code, change state and write new status into the old one.
	        IF (#t_UDT_Outfeed2StatesStatus.Specific.ChuteDisabled <> #s_UDT_Outfeed2StatesStatusOld.Specific.ChuteDisabled AND NOT #sx_SendAllProcedure)
	            OR (#sx_SendAllProcedure AND #ii_ErrorNumber = 0)
	        THEN
	            #sdi_Code := "DB_MFC_ErrorCode".Outfeed2States.ChuteDisabled;
	            #si_State := BOOL_TO_INT(#t_UDT_Outfeed2StatesStatus.Specific.ChuteDisabled);
	            #s_UDT_Outfeed2StatesStatusOld.Specific.ChuteDisabled := #t_UDT_Outfeed2StatesStatus.Specific.ChuteDisabled;
	            #sx_ItemErrorMessageReq := TRUE;
	            #ii_ErrorNumber += 1;
	        ELSIF (#t_UDT_Outfeed2StatesStatus.Specific.ChuteFull <> #s_UDT_Outfeed2StatesStatusOld.Specific.ChuteFull AND NOT #sx_SendAllProcedure)
	            OR (#sx_SendAllProcedure AND #ii_ErrorNumber = 1)
	        THEN
	            #sdi_Code := "DB_MFC_ErrorCode".Outfeed2States.ChuteFull;
	            #si_State := BOOL_TO_INT(#t_UDT_Outfeed2StatesStatus.Specific.ChuteFull);
	            #s_UDT_Outfeed2StatesStatusOld.Specific.ChuteFull := #t_UDT_Outfeed2StatesStatus.Specific.ChuteFull;
	            #sx_ItemErrorMessageReq := TRUE;
	            #ii_ErrorNumber += 1;
	        ELSIF (#t_UDT_Outfeed2StatesStatus.Specific.ChuteHalfFull <> #s_UDT_Outfeed2StatesStatusOld.Specific.ChuteHalfFull AND NOT #sx_SendAllProcedure)
	            OR (#sx_SendAllProcedure AND #ii_ErrorNumber = 2)
	        THEN
	            #sdi_Code := "DB_MFC_ErrorCode".Outfeed2States.ChuteHalfFull;
	            #si_State := BOOL_TO_INT(#t_UDT_Outfeed2StatesStatus.Specific.ChuteHalfFull);
	            #s_UDT_Outfeed2StatesStatusOld.Specific.ChuteHalfFull := #t_UDT_Outfeed2StatesStatus.Specific.ChuteHalfFull;
	            #sx_ItemErrorMessageReq := TRUE;
	            #sx_SendAllProcedure := FALSE;
	            #ii_ErrorNumber += 1;
	        END_IF;



	    END_IF;
	END_REGION

	REGION 4 - Write message components to the item error structure

	    #s_UDT_ItemError.ItemNumber := #i_UDT_EquipmentNumber;
	    #s_UDT_ItemError.Error := #sdi_Code;
	    #s_UDT_ItemError.State := #si_State;
	    #s_UDT_ItemError.Masked := 1;

	END_REGION

	REGION 5 - Write message components to the item status structure

	    #s_UDT_ItemStatus.Group := #i_UDT_EquipmentNumber.Group;
	    #s_UDT_ItemStatus.Node := #i_UDT_EquipmentNumber.Node;
	    #s_UDT_ItemStatus.Status := #si_ItemStatus;

	END_REGION

	REGION 6 - Prepare messages to the MFC

	    // If item error message required signal is set, prepare the item error message.
	    IF (#sx_ItemErrorMessageReq)
	    THEN
	        #s_FB_ItemError(i_UDT_ItemErrorBody := #s_UDT_ItemError,
	                        ii_MessageGroup := 1,
	                        ix_FlagRetry := FALSE,
	                        idi_TimeSpan := 0,
	                        qx_Error => #sx_ItemErrorBlockError,
	                        qx_Warning => #sx_ItemErrorBlockWarning,
	                        iq_UDT_FifoHeader := #iq_UDT_FifoHeader,
	                        iqs_FifoData := #iqs_FifoData,
	                        iqdi_MessageSequenceNumber := #iqdi_MessageSequenceNumber);
	    END_IF;

	    // If item status message required signal is set, prepare the item error message.
	    IF (#sx_ItemStatusMessageReq)
	    THEN
	        #s_FB_ItemStatus(i_UDT_ItemStatusBody := #s_UDT_ItemStatus,
	                         ii_MessageGroup := 1,
	                         ix_FlagRetry := FALSE,
	                         idi_TimeSpan := 0,
	                         qx_Error => #sx_ItemStatusBlockError,
	                         qx_Warning => #sx_ItemStatusBlockWarning,
	                         iq_UDT_FifoHeader := #iq_UDT_FifoHeader,
	                         iqs_FifoData := #iqs_FifoData,
	                         iqdi_MessageSequenceNumber := #iqdi_MessageSequenceNumber);
	    END_IF;

	END_REGION

	REGION 7 - Write outputs

	    // Prepare collective output error.
	    #qx_Error :=
	    #sx_ItemErrorBlockError
	    OR #sx_ItemStatusBlockError
	    OR #sx_FIFOError;

	    // Prepare collective output warning.
	    #qx_Warning :=
	    #sx_ItemErrorBlockWarning
	    OR #sx_ItemStatusBlockWarning
	    OR #sx_FIFOWarning;

	END_REGION
END_FUNCTION_BLOCK

FUNCTION_BLOCK "FB_MFC_Visu_TCPIPConncetion_Status"
{ S7_Optimized_Access := 'TRUE' }
VERSION : 0.1
// ATTRIBUTES
// AUTO_NUMBER = True
// BLOCK_NUMBER = 160
// END_ATTRIBUTES
   VAR_INPUT
      i_UDT_TCPIPConnectStatus { ExternalAccessible := 'False'; ExternalVisible := 'False'; ExternalWritable := 'False'} : "UDT_TCPIPConnectStatus";   // TCPIPConnection status structure
      i_UDT_EquipmentNumber { ExternalAccessible := 'False'; ExternalVisible := 'False'; ExternalWritable := 'False'} : "UDT_EquipmentNumber";   // Item number
      ix_SendAllErrorsState { ExternalAccessible := 'False'; ExternalVisible := 'False'; ExternalWritable := 'False'} : Bool;   // True - update all the messages
      ix_MFCConnected { ExternalAccessible := 'False'; ExternalVisible := 'False'; ExternalWritable := 'False'} : Bool;   // True - A connection to the MFC has been established
      ix_CollectiveReset { ExternalAccessible := 'False'; ExternalVisible := 'False'; ExternalWritable := 'False'} : Bool;   // True - Collective reset command of all system controls
   END_VAR

   VAR_OUTPUT
      qx_Error { ExternalAccessible := 'False'; ExternalVisible := 'False'; ExternalWritable := 'False'} : Bool;   // Block error
      qx_Warning { ExternalAccessible := 'False'; ExternalVisible := 'False'; ExternalWritable := 'False'} : Bool;   // Block warning
   END_VAR

   VAR_IN_OUT
      iq_UDT_FifoHeader : "UDT_FifoHeader";   // FIFO header
      iqs_FifoData : Array[*] of "UDT_MessageV2";   // FIFO data buffer
      iqdi_MessageSequenceNumber { ExternalAccessible := 'False'; ExternalVisible := 'False'; ExternalWritable := 'False'} : DInt;   // Message number
   END_VAR

   VAR
      s_FB_ItemError { ExternalAccessible := 'False'; ExternalVisible := 'False'; ExternalWritable := 'False'; S7_SetPoint := 'False'} : "FB_ItemError";   // Item error block's instance
      s_FB_ItemStatus { ExternalAccessible := 'False'; ExternalVisible := 'False'; ExternalWritable := 'False'; S7_SetPoint := 'False'} : "FB_ItemStatus";   // Item status block's instance
      ss_FIFOStatus { ExternalAccessible := 'False'; ExternalVisible := 'False'; ExternalWritable := 'False'; S7_SetPoint := 'False'} : "UDT_FifoStatus";   // Status structure
      s_UDT_Message { ExternalAccessible := 'False'; ExternalVisible := 'False'; ExternalWritable := 'False'; S7_SetPoint := 'False'} : "UDT_MessageV2";   // Message
      s_UDT_TCPIPConnectStatusOld { ExternalAccessible := 'False'; ExternalVisible := 'False'; ExternalWritable := 'False'; S7_SetPoint := 'False'} : "UDT_TCPIPConnectStatus";   // TCPIPConnection status structure
      s_UDT_ItemError { ExternalAccessible := 'False'; ExternalVisible := 'False'; ExternalWritable := 'False'; S7_SetPoint := 'False'} : "UDT_ItemError";   // Item error message body structure
      s_UDT_ItemStatus { ExternalAccessible := 'False'; ExternalVisible := 'False'; ExternalWritable := 'False'; S7_SetPoint := 'False'} : "UDT_ItemStatus";   // Item status message body structure
      s_R_TRIG_Connection {InstructionName := 'R_TRIG'; LibVersion := '1.0'; ExternalAccessible := 'False'; ExternalVisible := 'False'; ExternalWritable := 'False'; S7_SetPoint := 'False'} : R_TRIG;   // Rising edge trigger connection reastablished
      s_F_TRIG_SendAllErrors {InstructionName := 'F_TRIG'; LibVersion := '1.0'; ExternalAccessible := 'False'; ExternalVisible := 'False'; ExternalWritable := 'False'; S7_SetPoint := 'False'} : F_TRIG;   // Falling edge trigger from signal send all errors
      sdi_Code { ExternalAccessible := 'False'; ExternalVisible := 'False'; ExternalWritable := 'False'} : DInt;   // Error code
      si_ItemStatus { ExternalAccessible := 'False'; ExternalVisible := 'False'; ExternalWritable := 'False'} : Int;   // Item status
      ii_ErrorNumber { ExternalAccessible := 'False'; ExternalVisible := 'False'; ExternalWritable := 'False'} : Int;   // Counter Error Number
      si_State { ExternalAccessible := 'False'; ExternalVisible := 'False'; ExternalWritable := 'False'} : Int;   // Error state
      sx_ItemErrorMessageReq { ExternalAccessible := 'False'; ExternalVisible := 'False'; ExternalWritable := 'False'} : Bool;   // Item error message required
      sx_ItemStatusMessageReq { ExternalAccessible := 'False'; ExternalVisible := 'False'; ExternalWritable := 'False'} : Bool;   // Item status message required
      sx_SendAllProcedure { ExternalAccessible := 'False'; ExternalVisible := 'False'; ExternalWritable := 'False'} : Bool;   // Send all procedure
      sx_FIFOError { ExternalAccessible := 'False'; ExternalVisible := 'False'; ExternalWritable := 'False'} : Bool;   // FIFO error
      sx_FIFOWarning { ExternalAccessible := 'False'; ExternalVisible := 'False'; ExternalWritable := 'False'} : Bool;   // FIFO warning
      sx_ItemErrorBlockError { ExternalAccessible := 'False'; ExternalVisible := 'False'; ExternalWritable := 'False'} : Bool;   // Item error block error
      sx_ItemErrorBlockWarning { ExternalAccessible := 'False'; ExternalVisible := 'False'; ExternalWritable := 'False'} : Bool;   // Item error block warning
      sx_ItemStatusBlockError { ExternalAccessible := 'False'; ExternalVisible := 'False'; ExternalWritable := 'False'} : Bool;   // Item status block error
      sx_ItemStatusBlockWarning { ExternalAccessible := 'False'; ExternalVisible := 'False'; ExternalWritable := 'False'} : Bool;   // Item status block warning
   END_VAR


BEGIN
	(*
	----------------------------------------------------------------------------------------
	|                                                                                      |
	|  Copyright  2023             FORTNA Europe BV                                        |
	|  All Rights Reserved         Netherlands                                             |
	|                                                                                      |
	----------------------------------------------------------------------------------------
	Version history:
	Date        | Version   | Author       | Remark
	----------------------------------------------------------------------------------------
	24/03/2023  | 1.0       | M. Diebel   | Release TIA 17 | DHL Munich 2023
	13/03/2023  | 1.1       | S. Nieswiec  | Updated for new Baseline
	*)


	REGION 1 - Initialize message required signals

	    #sx_ItemErrorMessageReq := FALSE;
	    #sx_ItemStatusMessageReq := FALSE;

	    // On connection reestablish send last remembered status and error state ( status only when it's diffrent then 0 )
	    #s_R_TRIG_Connection(CLK := #ix_MFCConnected);

	    IF #s_R_TRIG_Connection.Q AND #si_ItemStatus <> 0
	    THEN
	        #sx_ItemStatusMessageReq := TRUE;
	    END_IF;

	    IF #s_R_TRIG_Connection.Q
	    THEN
	        #sx_ItemErrorMessageReq := TRUE;
	    END_IF;

	    // Prepare trigger on the collective reset signal.
	    #s_F_TRIG_SendAllErrors(CLK := #ix_SendAllErrorsState);

	    // When collective reset will go down, start send every equipment errors.
	    IF #s_F_TRIG_SendAllErrors.Q AND NOT #sx_SendAllProcedure
	    THEN
	        #ii_ErrorNumber := 0;
	        #sx_SendAllProcedure := TRUE;
	    END_IF;

	END_REGION

	REGION 2 - FIFO header status update

	    // Mode 'S' - FIFO register status update.
	    "FC_Fifo"(ic_Mode := 'S',
	              qUDT_Status => #ss_FIFOStatus,
	              qx_Error => #sx_FIFOError,
	              qx_Warning => #sx_FIFOWarning,
	              iqv_Data := #s_UDT_Message,
	              iqUDT_FifoHeader := #iq_UDT_FifoHeader,
	              iqv_DataBuffer := #iqs_FifoData);

	END_REGION

	REGION 3 - Prepare message data

	    // When there is no reset errors command, update status and errors.
	    IF NOT #ix_CollectiveReset
	        AND NOT #ss_FIFOStatus.FifoPreFull
	    THEN
	        // Status
	        IF (#i_UDT_TCPIPConnectStatus.Status <> #s_UDT_TCPIPConnectStatusOld.Status OR (#sx_SendAllProcedure AND #ii_ErrorNumber = 0))
	        THEN
	            #sx_ItemStatusMessageReq := TRUE;
	            #si_ItemStatus := #i_UDT_TCPIPConnectStatus.Status;
	            #s_UDT_TCPIPConnectStatusOld.Status := #i_UDT_TCPIPConnectStatus.Status;
	        END_IF;


	        // Check which specific status changed, prepare code, change state and write new status into the old one.
	        IF (#i_UDT_TCPIPConnectStatus.Specific.CommunicationFault <> #s_UDT_TCPIPConnectStatusOld.Specific.CommunicationFault AND NOT #sx_SendAllProcedure)
	            OR (#sx_SendAllProcedure AND #ii_ErrorNumber = 0)
	        THEN
	            #sdi_Code := "DB_MFC_ErrorCode".TCPIPConnection.CommunicationFault;
	            #si_State := BOOL_TO_INT(#i_UDT_TCPIPConnectStatus.Specific.CommunicationFault);
	            #s_UDT_TCPIPConnectStatusOld.Specific.CommunicationFault := #i_UDT_TCPIPConnectStatus.Specific.CommunicationFault;
	            #sx_ItemErrorMessageReq := TRUE;
	            #sx_SendAllProcedure := FALSE;
	        END_IF;
	    END_IF;
	END_REGION

	REGION 4 - Write message components to the item error structure

	    #s_UDT_ItemError.ItemNumber := #i_UDT_EquipmentNumber;
	    #s_UDT_ItemError.Error := #sdi_Code;
	    #s_UDT_ItemError.State := #si_State;
	    #s_UDT_ItemError.Masked := 1;

	END_REGION

	REGION 5 - Write message components to the item status structure

	    #s_UDT_ItemStatus.Group := #i_UDT_EquipmentNumber.Group;
	    #s_UDT_ItemStatus.Node := #i_UDT_EquipmentNumber.Node;
	    #s_UDT_ItemStatus.Status := #si_ItemStatus;

	END_REGION

	REGION 6 - Prepare messages to the MFC

	    // If item error message required signal is set, prepare the item error message.
	    IF (#sx_ItemErrorMessageReq)
	    THEN
	        #s_FB_ItemError(i_UDT_ItemErrorBody := #s_UDT_ItemError,
	                        ii_MessageGroup := 1,
	                        ix_FlagRetry := FALSE,
	                        idi_TimeSpan := 0,
	                        qx_Error => #sx_ItemErrorBlockError,
	                        qx_Warning => #sx_ItemErrorBlockWarning,
	                        iq_UDT_FifoHeader := #iq_UDT_FifoHeader,
	                        iqs_FifoData := #iqs_FifoData,
	                        iqdi_MessageSequenceNumber := #iqdi_MessageSequenceNumber);
	    END_IF;

	    // If item status message required signal is set, prepare the item error message.
	    IF (#sx_ItemStatusMessageReq)
	    THEN
	        #s_FB_ItemStatus(i_UDT_ItemStatusBody := #s_UDT_ItemStatus,
	                         ii_MessageGroup := 1,
	                         ix_FlagRetry := FALSE,
	                         idi_TimeSpan := 0,
	                         qx_Error => #sx_ItemStatusBlockError,
	                         qx_Warning => #sx_ItemStatusBlockWarning,
	                         iq_UDT_FifoHeader := #iq_UDT_FifoHeader,
	                         iqs_FifoData := #iqs_FifoData,
	                         iqdi_MessageSequenceNumber := #iqdi_MessageSequenceNumber);
	    END_IF;

	END_REGION

	REGION 7 - Write outputs

	    // Prepare collective output error.
	    #qx_Error :=
	    #sx_ItemErrorBlockError
	    OR #sx_ItemStatusBlockError
	    OR #sx_FIFOError;

	    // Prepare collective output warning.
	    #qx_Warning :=
	    #sx_ItemErrorBlockWarning
	    OR #sx_ItemStatusBlockWarning
	    OR #sx_FIFOWarning;

	END_REGION




END_FUNCTION_BLOCK

FUNCTION_BLOCK "FB_MFC_Visu_PDP_Status"
{ S7_Optimized_Access := 'TRUE' }
VERSION : 1.1
// ATTRIBUTES
// AUTO_NUMBER = True
// BLOCK_NUMBER = 153
// END_ATTRIBUTES
   VAR_INPUT
      i_UDT_PDPStatus { ExternalAccessible := 'False'; ExternalVisible := 'False'; ExternalWritable := 'False'} : "UDT_PDPStatus";
      i_UDT_EquipmentNumber { ExternalAccessible := 'False'; ExternalVisible := 'False'; ExternalWritable := 'False'} : "UDT_EquipmentNumber";   // Item number
      ix_SendAllErrorsState { ExternalAccessible := 'False'; ExternalVisible := 'False'; ExternalWritable := 'False'} : Bool;   // True - update all the messages
      ix_MFCConnected { ExternalAccessible := 'False'; ExternalVisible := 'False'; ExternalWritable := 'False'} : Bool;   // True - A connection to the MFC has been established
      ix_CollectiveReset { ExternalAccessible := 'False'; ExternalVisible := 'False'; ExternalWritable := 'False'} : Bool;   // True - Collective reset command of all system controls
   END_VAR

   VAR_OUTPUT
      qx_Error { ExternalAccessible := 'False'; ExternalVisible := 'False'; ExternalWritable := 'False'} : Bool;   // Block error
      qx_Warning { ExternalAccessible := 'False'; ExternalVisible := 'False'; ExternalWritable := 'False'} : Bool;   // Block warning
   END_VAR

   VAR_IN_OUT
      iq_UDT_FifoHeader : "UDT_FifoHeader";   // FIFO header
      iqs_FifoData : Array[*] of "UDT_MessageV2";   // FIFO data buffer
      iqdi_MessageSequenceNumber { ExternalAccessible := 'False'; ExternalVisible := 'False'; ExternalWritable := 'False'} : DInt;   // Message number
   END_VAR

   VAR
      s_FB_ItemStatus { ExternalAccessible := 'False'; ExternalVisible := 'False'; ExternalWritable := 'False'; S7_SetPoint := 'False'} : "FB_ItemStatus";   // Item status block's instance
      s_FB_ItemError { ExternalAccessible := 'False'; ExternalVisible := 'False'; ExternalWritable := 'False'; S7_SetPoint := 'False'} : "FB_ItemError";   // Item error block's instance
      s_UDT_ItemStatus { ExternalAccessible := 'False'; ExternalVisible := 'False'; ExternalWritable := 'False'; S7_SetPoint := 'False'} : "UDT_ItemStatus";   // Item status message body structure
      ss_FIFOStatus { ExternalAccessible := 'False'; ExternalVisible := 'False'; ExternalWritable := 'False'; S7_SetPoint := 'False'} : "UDT_FifoStatus";   // Status structure
      s_UDT_Message { ExternalAccessible := 'False'; ExternalVisible := 'False'; ExternalWritable := 'False'; S7_SetPoint := 'False'} : "UDT_MessageV2";   // Message
      s_UDT_PDPOldStatus { ExternalAccessible := 'False'; ExternalVisible := 'False'; ExternalWritable := 'False'; S7_SetPoint := 'False'} : "UDT_PDPStatus";
      s_UDT_ItemError { ExternalAccessible := 'False'; ExternalVisible := 'False'; ExternalWritable := 'False'; S7_SetPoint := 'False'} : "UDT_ItemError";   // Item error message body structure
      s_R_TRIG_Connection {InstructionName := 'R_TRIG'; LibVersion := '1.0'; ExternalAccessible := 'False'; ExternalVisible := 'False'; ExternalWritable := 'False'; S7_SetPoint := 'False'} : R_TRIG;   // Rising edge trigger connection reastablished
      s_F_TRIG_SendAllErrors {InstructionName := 'F_TRIG'; LibVersion := '1.0'; ExternalAccessible := 'False'; ExternalVisible := 'False'; ExternalWritable := 'False'; S7_SetPoint := 'False'} : F_TRIG;   // Falling edge trigger from signal send all errors
      sdi_Code { ExternalAccessible := 'False'; ExternalVisible := 'False'; ExternalWritable := 'False'} : DInt;   // Error code
      si_ItemStatus { ExternalAccessible := 'False'; ExternalVisible := 'False'; ExternalWritable := 'False'} : Int;   // Item status
      ii_ErrorNumber { ExternalAccessible := 'False'; ExternalVisible := 'False'; ExternalWritable := 'False'} : Int;   // Counter Error Number
      si_State { ExternalAccessible := 'False'; ExternalVisible := 'False'; ExternalWritable := 'False'} : Int;   // Error state
      sx_ItemErrorMessageReq { ExternalAccessible := 'False'; ExternalVisible := 'False'; ExternalWritable := 'False'} : Bool;   // Item error message required
      sx_ItemStatusMessageReq { ExternalAccessible := 'False'; ExternalVisible := 'False'; ExternalWritable := 'False'} : Bool;   // Item status message required
      sx_SendAllProcedure { ExternalAccessible := 'False'; ExternalVisible := 'False'; ExternalWritable := 'False'} : Bool;   // Send all procedure
      sx_FIFOError { ExternalAccessible := 'False'; ExternalVisible := 'False'; ExternalWritable := 'False'} : Bool;   // FIFO error
      sx_FIFOWarning { ExternalAccessible := 'False'; ExternalVisible := 'False'; ExternalWritable := 'False'} : Bool;   // FIFO warning
      sx_ItemErrorBlockError { ExternalAccessible := 'False'; ExternalVisible := 'False'; ExternalWritable := 'False'} : Bool;   // Item error block error
      sx_ItemErrorBlockWarning { ExternalAccessible := 'False'; ExternalVisible := 'False'; ExternalWritable := 'False'} : Bool;   // Item error block warning
      sx_ItemStatusBlockError { ExternalAccessible := 'False'; ExternalVisible := 'False'; ExternalWritable := 'False'} : Bool;   // Item status block error
      sx_ItemStatusBlockWarning { ExternalAccessible := 'False'; ExternalVisible := 'False'; ExternalWritable := 'False'} : Bool;   // Item status block warning
   END_VAR


BEGIN
	(*
	----------------------------------------------------------------------------------------
	|                                                                                      |
	|  Copyright  2023             FORTNA Europe BV                                        |
	|  All Rights Reserved         Netherlands                                             |
	|                                                                                      |
	----------------------------------------------------------------------------------------
	Version history:
	Date        | Version   | Author       | Remark
	----------------------------------------------------------------------------------------
	20/04/2023  | 1.0       | M. Diebel   | Release TIA 17 | DHL Munich 2023
	16/08/2023  | 1.1       | S. Theocharis| update with new PDP status
	13/03/2023  | 1.2       | S. Nieswiec  | Updated for new Baseline
	*)




	REGION 1 - Initialize message required signals

	    #sx_ItemErrorMessageReq := FALSE;
	    #sx_ItemStatusMessageReq := FALSE;

	    // On connection reestablish send last remembered status and error state ( status only when it's diffrent then 0 )
	    #s_R_TRIG_Connection(CLK := #ix_MFCConnected);

	    IF #s_R_TRIG_Connection.Q AND #si_ItemStatus <> 0
	    THEN
	        #sx_ItemStatusMessageReq := TRUE;
	    END_IF;

	    IF #s_R_TRIG_Connection.Q
	    THEN
	        #sx_ItemErrorMessageReq := TRUE;
	    END_IF;

	    // Prepare trigger on the collective reset signal.
	    #s_F_TRIG_SendAllErrors(CLK := #ix_SendAllErrorsState);

	    // When collective reset will go down, start send every equipment errors.
	    IF #s_F_TRIG_SendAllErrors.Q AND NOT #sx_SendAllProcedure
	    THEN
	        #ii_ErrorNumber := 0;
	        #sx_SendAllProcedure := TRUE;
	    END_IF;

	END_REGION

	REGION 2 - FIFO header status update

	    // Mode 'S' - FIFO register status update.
	    "FC_Fifo"(ic_Mode := 'S',
	              qUDT_Status => #ss_FIFOStatus,
	              qx_Error => #sx_FIFOError,
	              qx_Warning => #sx_FIFOWarning,
	              iqv_Data := #s_UDT_Message,
	              iqUDT_FifoHeader := #iq_UDT_FifoHeader,
	              iqv_DataBuffer := #iqs_FifoData);

	END_REGION

	REGION 3 - Prepare message data

	    // When there is no reset errors command, update status and errors.
	    IF NOT #ix_CollectiveReset
	        AND NOT #ss_FIFOStatus.FifoPreFull
	    THEN

	        // Status
	        IF (#i_UDT_PDPStatus.Status <> #s_UDT_PDPOldStatus.Status OR (#sx_SendAllProcedure AND #ii_ErrorNumber = 0))
	        THEN
	            #sx_ItemStatusMessageReq := TRUE;
	            #si_ItemStatus := #i_UDT_PDPStatus.Status;
	            #s_UDT_PDPOldStatus.Status := #i_UDT_PDPStatus.Status;
	        END_IF;


	        // Check which specific status changed, prepare code, change state and write new status into the old one.
	        IF (#i_UDT_PDPStatus.Specific.CircuitBreakersTripped <> #s_UDT_PDPOldStatus.Specific.CircuitBreakersTripped AND NOT #sx_SendAllProcedure)
	            OR (#sx_SendAllProcedure AND #ii_ErrorNumber = 0)
	        THEN
	            #sdi_Code := "DB_MFC_ErrorCode".PDP.CircuitBreakersTripped;
	            #si_State := BOOL_TO_INT(#i_UDT_PDPStatus.Specific.CircuitBreakersTripped);
	            #s_UDT_PDPOldStatus.Specific.CircuitBreakersTripped := #i_UDT_PDPStatus.Specific.CircuitBreakersTripped;
	            #sx_ItemErrorMessageReq := TRUE;
	            #ii_ErrorNumber += 1;
	        ELSIF (#i_UDT_PDPStatus.Specific.CircuitBreakerStateF100_F200_F300 <> #s_UDT_PDPOldStatus.Specific.CircuitBreakerStateF100_F200_F300 AND NOT #sx_SendAllProcedure)
	            OR (#sx_SendAllProcedure AND #ii_ErrorNumber = 1)
	        THEN
	            #sdi_Code := "DB_MFC_ErrorCode".PDP.CircuitBreakerStateF100_F200_F300;
	            #si_State := BOOL_TO_INT(#i_UDT_PDPStatus.Specific.CircuitBreakerStateF100_F200_F300);
	            #s_UDT_PDPOldStatus.Specific.CircuitBreakerStateF100_F200_F300 := #i_UDT_PDPStatus.Specific.CircuitBreakerStateF100_F200_F300;
	            #sx_ItemErrorMessageReq := TRUE;
	            #ii_ErrorNumber += 1;
	        ELSIF (#i_UDT_PDPStatus.Specific.CircuitBreakerStatePM <> #s_UDT_PDPOldStatus.Specific.CircuitBreakerStatePM AND NOT #sx_SendAllProcedure)
	            OR (#sx_SendAllProcedure AND #ii_ErrorNumber = 2)
	        THEN
	            #sdi_Code := "DB_MFC_ErrorCode".PDP.CircuitBreakerStatePM;
	            #si_State := BOOL_TO_INT(#i_UDT_PDPStatus.Specific.CircuitBreakerStatePM);
	            #s_UDT_PDPOldStatus.Specific.CircuitBreakerStatePM := #i_UDT_PDPStatus.Specific.CircuitBreakerStatePM;
	            #sx_ItemErrorMessageReq := TRUE;
	            #ii_ErrorNumber += 1;
	        ELSIF (#i_UDT_PDPStatus.Specific.CircuitBreakerTrippedF101 <> #s_UDT_PDPOldStatus.Specific.CircuitBreakerTrippedF101 AND NOT #sx_SendAllProcedure)
	            OR (#sx_SendAllProcedure AND #ii_ErrorNumber = 3)
	        THEN
	            #sdi_Code := "DB_MFC_ErrorCode".PDP.CircuitBreakerTrippedF101;
	            #si_State := BOOL_TO_INT(#i_UDT_PDPStatus.Specific.CircuitBreakerTrippedF101);
	            #s_UDT_PDPOldStatus.Specific.CircuitBreakerTrippedF101 := #i_UDT_PDPStatus.Specific.CircuitBreakerTrippedF101;
	            #sx_ItemErrorMessageReq := TRUE;
	            #ii_ErrorNumber += 1;



	        ELSIF (#i_UDT_PDPStatus.Specific.CircuitBreakerTrippedF102 <> #s_UDT_PDPOldStatus.Specific.CircuitBreakerTrippedF102 AND NOT #sx_SendAllProcedure)
	            OR (#sx_SendAllProcedure AND #ii_ErrorNumber = 4)
	        THEN
	            #sdi_Code := "DB_MFC_ErrorCode".PDP.CircuitBreakerTrippedF102;
	            #si_State := BOOL_TO_INT(#i_UDT_PDPStatus.Specific.CircuitBreakerTrippedF102);
	            #s_UDT_PDPOldStatus.Specific.CircuitBreakerTrippedF102 := #i_UDT_PDPStatus.Specific.CircuitBreakerTrippedF102;
	            #sx_ItemErrorMessageReq := TRUE;
	            #ii_ErrorNumber += 1;
	        ELSIF (#i_UDT_PDPStatus.Specific.CircuitBreakerTrippedF103 <> #s_UDT_PDPOldStatus.Specific.CircuitBreakerTrippedF103 AND NOT #sx_SendAllProcedure)
	            OR (#sx_SendAllProcedure AND #ii_ErrorNumber = 5)
	        THEN
	            #sdi_Code := "DB_MFC_ErrorCode".PDP.CircuitBreakerTrippedF103;
	            #si_State := BOOL_TO_INT(#i_UDT_PDPStatus.Specific.CircuitBreakerTrippedF103);
	            #s_UDT_PDPOldStatus.Specific.CircuitBreakerTrippedF103 := #i_UDT_PDPStatus.Specific.CircuitBreakerTrippedF103;
	            #sx_ItemErrorMessageReq := TRUE;
	            #ii_ErrorNumber += 1;
	        ELSIF (#i_UDT_PDPStatus.Specific.CircuitBreakerTrippedF104 <> #s_UDT_PDPOldStatus.Specific.CircuitBreakerTrippedF104 AND NOT #sx_SendAllProcedure)
	            OR (#sx_SendAllProcedure AND #ii_ErrorNumber = 6)
	        THEN
	            #sdi_Code := "DB_MFC_ErrorCode".PDP.CircuitBreakerTrippedF104;
	            #si_State := BOOL_TO_INT(#i_UDT_PDPStatus.Specific.CircuitBreakerTrippedF104);
	            #s_UDT_PDPOldStatus.Specific.CircuitBreakerTrippedF104 := #i_UDT_PDPStatus.Specific.CircuitBreakerTrippedF104;
	            #sx_ItemErrorMessageReq := TRUE;
	            #ii_ErrorNumber += 1;
	        ELSIF (#i_UDT_PDPStatus.Specific.CircuitBreakerTrippedF105 <> #s_UDT_PDPOldStatus.Specific.CircuitBreakerTrippedF105 AND NOT #sx_SendAllProcedure)
	            OR (#sx_SendAllProcedure AND #ii_ErrorNumber = 7)
	        THEN
	            #sdi_Code := "DB_MFC_ErrorCode".PDP.CircuitBreakerTrippedF105;
	            #si_State := BOOL_TO_INT(#i_UDT_PDPStatus.Specific.CircuitBreakerTrippedF105);
	            #s_UDT_PDPOldStatus.Specific.CircuitBreakerTrippedF105 := #i_UDT_PDPStatus.Specific.CircuitBreakerTrippedF105;
	            #sx_ItemErrorMessageReq := TRUE;
	            #ii_ErrorNumber += 1;
	        ELSIF (#i_UDT_PDPStatus.Specific.CircuitBreakerTrippedF106 <> #s_UDT_PDPOldStatus.Specific.CircuitBreakerTrippedF106 AND NOT #sx_SendAllProcedure)
	            OR (#sx_SendAllProcedure AND #ii_ErrorNumber = 8)
	        THEN
	            #sdi_Code := "DB_MFC_ErrorCode".PDP.CircuitBreakerTrippedF106;
	            #si_State := BOOL_TO_INT(#i_UDT_PDPStatus.Specific.CircuitBreakerTrippedF106);
	            #s_UDT_PDPOldStatus.Specific.CircuitBreakerTrippedF106 := #i_UDT_PDPStatus.Specific.CircuitBreakerTrippedF106;
	            #sx_ItemErrorMessageReq := TRUE;
	            #ii_ErrorNumber += 1;
	        ELSIF (#i_UDT_PDPStatus.Specific.CircuitBreakerTrippedF107 <> #s_UDT_PDPOldStatus.Specific.CircuitBreakerTrippedF107 AND NOT #sx_SendAllProcedure)
	            OR (#sx_SendAllProcedure AND #ii_ErrorNumber = 9)
	        THEN
	            #sdi_Code := "DB_MFC_ErrorCode".PDP.CircuitBreakerTrippedF107;
	            #si_State := BOOL_TO_INT(#i_UDT_PDPStatus.Specific.CircuitBreakerTrippedF107);
	            #s_UDT_PDPOldStatus.Specific.CircuitBreakerTrippedF107 := #i_UDT_PDPStatus.Specific.CircuitBreakerTrippedF107;
	            #sx_ItemErrorMessageReq := TRUE;
	            #ii_ErrorNumber += 1;



